FUNCTION_BLOCK Crane EXTENDS BaseCarrier
VAR_INPUT
END_VAR
VAR_OUTPUT
	o_VacuumGripper: VacuumGripper;
	o_MonostableCylinder: MonostableCylinder;
	// the angle with limited knowledge, e.g., -1 before stack, +1 after stack, +89 before LSC, +91 after LSC etc.
	o_Angle: INT := 45;
END_VAR
VAR
	// Turning table
	m_PresenceSensorAtStack : PresenceSensor;
	m_PresenceSensorAtConveyor : PresenceSensor;
	m_PresenceSensorAtStamp : PresenceSensor;
END_VAR

PROPERTY AtConveyor : BOOL
GET
AtConveyor := m_PresenceSensorAtConveyor.Value;
END_GET
END_PROPERTY

PROPERTY AtStack : BOOL
GET
AtStack := m_PresenceSensorAtStack.Value;
END_GET
END_PROPERTY

PROPERTY AtStamp : BOOL
GET
AtStamp := m_PresenceSensorAtStamp.Value;
END_GET
END_PROPERTY

METHOD METH_CarrierStop : BOOL
VAR_INPUT
END_VAR
Motor.ACT_Stop();
END_METHOD

METHOD METH_CarrierTurnClockwise : BOOL
VAR_INPUT
END_VAR
Motor.ACT_TurnClockwise();

IF AtStack THEN
	o_angle := 0;
ELSIF AtConveyor THEN
	o_angle := 90;
ELSIF AtStamp THEN
	o_angle := 180;
END_IF
END_METHOD

METHOD METH_CarrierTurnCounterclockwise : BOOL
VAR_INPUT
END_VAR
Motor.ACT_TurnCounterclockwise();

IF AtStack THEN
	o_angle := 0;
ELSIF AtConveyor THEN
	o_angle := 90;
ELSIF AtStamp THEN
	o_angle := 180;
END_IF
END_METHOD

END_FUNCTION_BLOCK

(* stored: Version 1.1.0.1, ProductVersion 3.1.4024.9
   POU Crane: Id {89659484-f4b6-4d4e-9769-13bb54647fd5}, SpecialFunc None
   Property AtConveyor: Id {98be1ca6-aaeb-4be7-a201-775c3d705d7f}
   Get Get: Id {ff456294-e1f9-4269-81bc-c634ad5bfbfe}
   Property AtStack: Id {d9e921f5-807a-447c-beb6-2f92290dbb0e}
   Get Get: Id {a2fd4aed-6330-4971-9d5e-16807bd877e9}
   Property AtStamp: Id {eb404776-4140-4f3b-817a-19497c2dc678}
   Get Get: Id {6e2f2f60-cdde-4232-b548-15b0f34b2c67}
   Method METH_CarrierStop: Id {af880bad-164b-4f34-8563-ba6d325f7c14}
   Method METH_CarrierTurnClockwise: Id {63741894-1719-4a74-9bdd-7facdefa00ba}
   Method METH_CarrierTurnCounterclockwise: Id {9d762642-289c-4e3d-803b-b09ea30dd23f} *)
